TYPE ST_BigBagDischargeInCmd :
STRUCT
    bEnable                 : BOOL;   // uruchomienie rozładunku
END_STRUCT
END_TYPE

(* stored: Version 1.1.0.1, ProductVersion 3.1.4024.16
   DUT ST_BigBagDischargeInCmd: Id {dea490ab-f2ab-4bb4-9340-fafb5ab7a2e3} *)
